TYPE ST_SoftSettings_Grid EXTENDS ST_SoftSettings_PeakshaveBox :
STRUCT
	b_GridCodesActive				: BOOL := TRUE;
	b_WeakGridInput					: BOOL;
	breaker							: ST_Input_breakersettings;
END_STRUCT
END_TYPE

(* stored: Version 1.1.0.1, ProductVersion 3.1.4026.18
   DUT ST_SoftSettings_Grid: Id {b7761e76-d30c-4be2-9254-25ad7acb1b31} *)
